PROGRAM PRG_LVCP1_CompensationCalculate
VAR
    fbCompensationCalc : FB_CompensationCalculator;
    bCalculate : BOOL := TRUE;              // Sürekli hesaplama için
    nActiveGroups : INT := 10;              // Toplam 10 grup
    
    // Outputs
    stHMIData : ST_CompensationHMI;
    asCapacitorTags : ARRAY[0..99] OF STRING(30);
    nActiveTags : INT;
    
    // Özet bilgiler
    rTotalPower : REAL;
    nTotalCapacitors : INT;
    nActiveGroupCount : INT;
END_VAR

// Grup sayısını güncelle
GVL_LVCP1.nConfiguredGroups := nActiveGroups;

// Hesaplama
fbCompensationCalc(
    bExecute 				:= bCalculate,
    bGroupActive 			:= GVL_LVCP1.abGroupActive,
    stGroupConfig 			:= GVL_LVCP1.astCompensationGroups,
    nActiveGroups 			:= GVL_LVCP1.nConfiguredGroups,
    stHMI 					=> stHMIData,
    asActiveCapacitorTags 	=> asCapacitorTags,
    nActiveCapacitorCount 	=> nActiveTags
);

// Özet bilgiler
rTotalPower 		:= stHMIData.stSummary.rTotalActivePower;
nTotalCapacitors 	:= stHMIData.stSummary.nTotalActiveCapacitors;
nActiveGroupCount 	:= stHMIData.stSummary.nActiveGroupCount;

END_PROGRAM

(* stored: Version 1.1.0.1, ProductVersion 3.1.4024.15
   POU PRG_LVCP1_CompensationCalculate: Id {ef69af31-59c1-4939-a1c3-3e4a39f6679c}, SpecialFunc None *)
